// TwinCAT 3 PLC project Lampara_PLC
// ProgramVersion: 3.1.4024.0
// libraries:
//   Tc2_Standard, * (Beckhoff Automation GmbH)
//   Tc2_System, * (Beckhoff Automation GmbH)
//   Tc3_Module, * (Beckhoff Automation GmbH)
//   VisuDialogs, * (System)
// project tree:
//   / GlobalTextList.TcGTLO, PlcTask.TcTTO, Visualization Manager.TcVMO (not stored)
//   POUs/IL/ FB_LamparaAsignada_IL.TcPOU, FB_LamparaComputada_IL.TcPOU, FB_LamparaConmutada_IL.TcPOU, FB_LamparaIntermitente_IL.TcPOU, FB_LamparaMemorizada_IL.TcPOU, FB_LamparaTemporizada_IL.TcPOU, FB_LamparaTemporizada_IL_2.TcPOU
//   POUs/LD/ FB_LamparaAsignada_LD.TcPOU, FB_LamparaComputada_LD.TcPOU, FB_LamparaConmutada_LD.TcPOU, FB_LamparaConmutada_LD_2.TcPOU, FB_LamparaIntermitente_LD.TcPOU, FB_LamparaMemorizada_LD.TcPOU, FB_LamparaMemorizada_LD_2.TcPOU, FB_LamparaTemporizada_LD.TcPOU, FB_LamparaTemporizada_LD_2.TcPOU
//   POUs/ MAIN.TcPOU
//   POUs/SFC/ FB_LamparaAsignada_SFC.TcPOU, FB_LamparaAsignada_SFC_2.TcPOU, FB_LamparaComputada_SFC.TcPOU, FB_LamparaConmutada_SFC.TcPOU, FB_LamparaConmutada_SFC_2.TcPOU, FB_LamparaIntermitente_SFC.TcPOU, FB_LamparaIntermitente_SFC_2.TcPOU, FB_LamparaMemorizada_SFC.TcPOU, FB_LamparaMemorizada_SFC_2.TcPOU, FB_LamparaTemporizada_SFC.TcPOU, FB_LamparaTemporizada_SFC_2.TcPOU
//   POUs/ST/ FB_LamparaAsignada_ST.TcPOU, FB_LamparaComputada_ST.TcPOU, FB_LamparaConmutada_ST.TcPOU, FB_LamparaIntermitente_ST.TcPOU, FB_LamparaMemorizada_ST.TcPOU, FB_LamparaTemporizada_ST.TcPOU, FB_LamparaTemporizada_ST_2.TcPOU, FB_LamparaTemporizada_ST_3.TcPOU
//   VISUs/ VISU_Lampara.TcVIS
// real-time tasks:
//   TASK PlcTask: cycle T#10ms, priority 20, ADS port 350
//   TASK PlcTask1: cycle T#10ms, priority 21, ADS port 351

CONFIGURATION Lampara_PLC
    RESOURCE PLC ON TwinCAT3
        TASK PlcTask(INTERVAL := T#10ms, PRIORITY := 20);
        PROGRAM MAIN WITH PlcTask : MAIN;
    END_RESOURCE
END_CONFIGURATION

// ---- POUs/MAIN.TcPOU
PROGRAM MAIN
(*
 * =================================================================================
 * POU Nombre:      MAIN
 * File:            MAIN.TcPOU
 * Version:         1.0.0
 * Date:            2025-10-20
 * Author:          Victor Torres
 * ---------------------------------------------------------------------------------
 * Copyright (C) 2020-2025 Victor Torres
 * License:         GNU General Public License (GPL)
 * This program is free software; see the file "LICENSE" for details
 * ---------------------------------------------------------------------------------
 * Historial de Revisiones:
 * ------------------------
 * 1.0.0 - 2025-10-20 - VTL: Versión inicial
 * 0.1.0 - 2020-05-02 - VTL: Creacion
 * =================================================================================
 *)
 
 (*!
 * @brief MAIN: Programa Principal de TC3_Lampara
 *
 * @description
 * Ejemplo sencillo para mostras el uso de los elementos fundamentales de la libreria 
 * STANDARD del IEC 61131-3 en los diferentes lenguajes de la norma.
 *
 * 1. Lampara asignada     - la lampara "copia" el estado del pulsador
 * 2. Lampara memoriazada  - un pulsador enciende la lampara y otro la apaga
 * 3. Lampara conmutada    - el mismo pulsador enciende y apaga la lampara
 * 4. Lampara temporizada  - la lampara se apaga transcurrido un cierto tiempo
 *                           despues de accionar el pulsador
 * 5. Lampara intermitente - la lampara parpadea
 * 6. Lampara computada    - la lampara se enciende tras accionar varias veces el 
 *                           pulsador y se apaga al accionar el pulsador de reinicio
*)
 
VAR
    Lampara   AT %Q*  : BOOL;
    Pulsador  AT %I*  : BOOL;
    
// Definir lo que corresponda {LENGUAJE_IL, LENGUAJE_LD, LENGUAJE_ST, LENGUAJE_SFC}
{define LENGUAJE_SFC}
{IF defined(LENGUAJE_IL)}
    LamparaAsignada      : FB_LamparaAsignada_IL;
    LamparaMemorizada    : FB_LamparaMemorizada_IL;
    LamparaConmutada     : FB_LamparaConmutada_IL;
    LamparaTemporizada   : FB_LamparaTemporizada_IL;
    LamparaIntermitente  : FB_LamparaIntermitente_IL;
    LamparaComputada     : FB_LamparaComputada_IL;
{ELSIF defined(LENGUAJE_LD)}
    LamparaAsignada      : FB_LamparaAsignada_LD;
    LamparaMemorizada    : FB_LamparaMemorizada_LD;
    LamparaConmutada     : FB_LamparaConmutada_LD;
    LamparaTemporizada   : FB_LamparaTemporizada_LD;
    LamparaIntermitente  : FB_LamparaIntermitente_LD;
    LamparaComputada     : FB_LamparaComputada_LD;
{ELSIF defined(LENGUAJE_ST)}
    LamparaAsignada      : FB_LamparaAsignada_ST;
    LamparaMemorizada    : FB_LamparaMemorizada_ST;
    LamparaConmutada     : FB_LamparaConmutada_ST;
    LamparaTemporizada   : FB_LamparaTemporizada_ST_3;
    LamparaIntermitente  : FB_LamparaIntermitente_ST;
    LamparaComputada     : FB_LamparaComputada_ST;
{ELSIF defined(LENGUAJE_SFC)}
    LamparaAsignada      : FB_LamparaAsignada_SFC;
    LamparaMemorizada    : FB_LamparaMemorizada_SFC;
    LamparaConmutada     : FB_LamparaConmutada_SFC;
    LamparaTemporizada   : FB_LamparaTemporizada_SFC;
    LamparaIntermitente  : FB_LamparaIntermitente_SFC_2;
    LamparaComputada     : FB_LamparaComputada_SFC;
{END_IF}
END_VAR

Lampara := Pulsador;

LamparaAsignada();
LamparaMemorizada();
LamparaConmutada();
LamparaTemporizada();
LamparaComputada();
LamparaIntermitente();

END_PROGRAM

// ---- POUs/IL/FB_LamparaAsignada_IL.TcPOU
FUNCTION_BLOCK FB_LamparaAsignada_IL
// La lampara se enciende mientras se acciona el pulsador
VAR
    Lampara   AT %Q*  : BOOL;
    Pulsador  AT %I*  : BOOL;
END_VAR

// NETWORK 1
// instruction list
LD      Pulsador
ST      Lampara

END_FUNCTION_BLOCK

// ---- POUs/IL/FB_LamparaMemorizada_IL.TcPOU
FUNCTION_BLOCK FB_LamparaMemorizada_IL
// La lampara se enciende al accionar el pulsador de conexion
// La lampara se apaga al accionar el pulsador de desconexion
VAR
    Lampara              AT %Q*  : BOOL;
    PulsadorConexion     AT %I*  : BOOL;
    PulsadorDesconexion  AT %I*  : BOOL;
END_VAR

// NETWORK 1
// instruction list
LD      PulsadorConexion
S       Lampara
LD      PulsadorDesconexion
R       Lampara

END_FUNCTION_BLOCK

// ---- POUs/IL/FB_LamparaConmutada_IL.TcPOU
FUNCTION_BLOCK FB_LamparaConmutada_IL
// La lampara se enciende si estando apagada se acciona el pulsador
// La lampara se apaga si estando encendida se acciona el pulsador
VAR
    Pulsacion         : R_TRIG;
    Lampara   AT %Q*  : BOOL;
    Pulsador  AT %I*  : BOOL;
END_VAR

// NETWORK 1
// instruction list
CAL     Pulsacion(
    CLK     := Pulsador)

// NETWORK 2
// instruction list
LD      Pulsacion.Q
JMPCN   End

// NETWORK 3
// instruction list
LDN     Lampara
ST      Lampara

// NETWORK 4
End:
// instruction list

END_FUNCTION_BLOCK

// ---- POUs/IL/FB_LamparaTemporizada_IL.TcPOU
FUNCTION_BLOCK FB_LamparaTemporizada_IL
// La lampara se enciende al accionar el pulsador
// La lampara se apaga transcurrido un tiempo encendidaVAR_INPUT
VAR
    TiempoEncendido   : TIME := T#2S;
END_VAR
VAR_OUTPUT
    TiempoPendiente   : TIME;
END_VAR
VAR
    Temporizador      : TON;
    Lampara   AT %Q*  : BOOL;
    Pulsador  AT %I*  : BOOL;
END_VAR

// NETWORK 1
// instruction list
CAL     Temporizador(
    IN      := Lampara,
    PT      := TiempoEncendido)

// NETWORK 2
// instruction list
LD      TiempoEncendido
SUB     Temporizador.ET
ST      TiempoPendiente

// NETWORK 3
// instruction list
LD      Pulsador
S       Lampara

// NETWORK 4
// instruction list
LD      Temporizador.Q
R       Lampara

END_FUNCTION_BLOCK

// ---- POUs/IL/FB_LamparaIntermitente_IL.TcPOU
FUNCTION_BLOCK FB_LamparaIntermitente_IL
// La lampara parpadea de forma continua
VAR_INPUT
    TiempoParpadeo   : TIME := T#500MS;
END_VAR
VAR
    Temporizador     : TON;
    Lampara  AT %Q*  : BOOL;
END_VAR

// NETWORK 1
// Temporizador auto-pilotado
// instruction list
CAL     Temporizador(
    IN      := NOT Temporizador.Q
    PT      := TiempoParpadeo)

// NETWORK 2
// instruction list
LD      Temporizador.Q
JMPCN   End

// NETWORK 3
// Salida conmutada
// instruction list
LD      Lampara
STN     Lampara

// NETWORK 4
End:
// instruction list

END_FUNCTION_BLOCK

// ---- POUs/IL/FB_LamparaComputada_IL.TcPOU
FUNCTION_BLOCK FB_LamparaComputada_IL
// La lampara se enciende tras un determinado numero de pulsaciones
// La lampara se apaga tras accionar el pulsador de reinicio
VAR_INPUT
    ManiobrasTotales     : UINT := 2;
END_VAR
VAR_OUTPUT
    ManiobrasPendientes  : UINT;
END_VAR
VAR
    Contador                  : CTD := (CV := ManiobrasTotales);
    Lampara           AT %Q*  : BOOL;
    Pulsador          AT %I*  : BOOL;
    PulsadorReinicio  AT %I*  : BOOL;
END_VAR

// NETWORK 1
// instruction list
CAL     Contador(
    CD      := Pulsador,
    LOAD    := PulsadorReinicio,
    PV      := ManiobrasTotales)

// NETWORK 2
// instruction list
LD      Contador.Q
ST      Lampara

// NETWORK 3
// instruction list
LD      Contador.CV
ST      ManiobrasPendientes

END_FUNCTION_BLOCK

// ---- POUs/LD/FB_LamparaAsignada_LD.TcPOU
FUNCTION_BLOCK FB_LamparaAsignada_LD
// La lampara se enciende mientras se acciona el pulsador
VAR
    Lampara   AT %Q*  : BOOL;
    Pulsador  AT %I*  : BOOL;
END_VAR

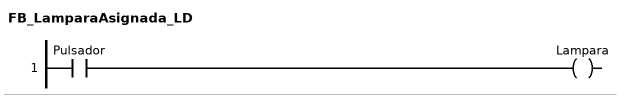
// NETWORK 1
Lampara := Pulsador;

END_FUNCTION_BLOCK

// ---- POUs/LD/FB_LamparaMemorizada_LD.TcPOU
FUNCTION_BLOCK FB_LamparaMemorizada_LD
// La lampara se enciende al accionar el pulsador de conexion
// La lampara se apaga al accionar el pulsador de desconexion
VAR
    Lampara              AT %Q*  : BOOL;
    PulsadorConexion     AT %I*  : BOOL;
    PulsadorDesconexion  AT %I*  : BOOL;
END_VAR

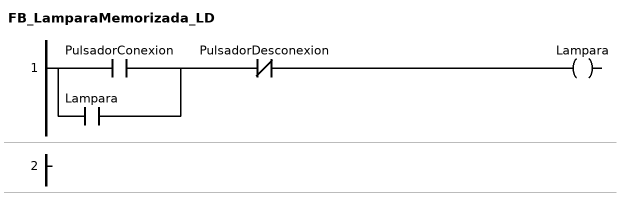
// NETWORK 1
Lampara := (PulsadorConexion OR Lampara) AND NOT PulsadorDesconexion;

// NETWORK 2

END_FUNCTION_BLOCK

// ---- POUs/LD/FB_LamparaConmutada_LD.TcPOU
FUNCTION_BLOCK FB_LamparaConmutada_LD
// La lampara se enciende si estando apagada se acciona el pulsador
// La lampara se apaga si estando encendida se acciona el pulsador
VAR
    Pulsacion         : R_TRIG;
    Lampara   AT %Q*  : BOOL;
    Pulsador  AT %I*  : BOOL;
END_VAR

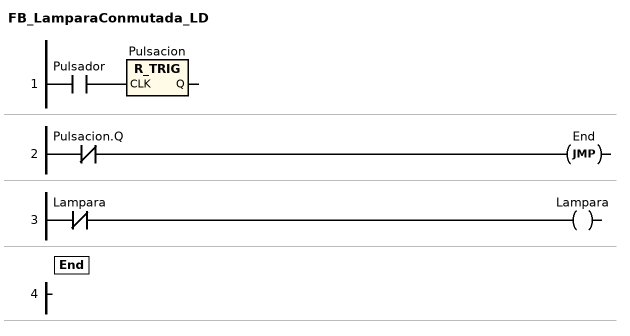
// NETWORK 1
Pulsacion(CLK := Pulsador); // R_TRIG

// NETWORK 2
IF NOT Pulsacion.Q THEN JMP End; END_IF

// NETWORK 3
Lampara := NOT Lampara;

// NETWORK 4
End: ;

END_FUNCTION_BLOCK

// ---- POUs/LD/FB_LamparaTemporizada_LD.TcPOU
FUNCTION_BLOCK FB_LamparaTemporizada_LD
// La lampara se enciende al accionar el pulsador
// La lampara se apaga transcurrido un tiempo encendida
VAR_INPUT
    TiempoEncendido   : TIME := T#2S;
END_VAR
VAR_OUTPUT
    TiempoPendiente   : TIME;
END_VAR
VAR
    Temporizador      : TON;
    Memoria           : RS;
    Lampara   AT %Q*  : BOOL;
    Pulsador  AT %I*  : BOOL;
END_VAR

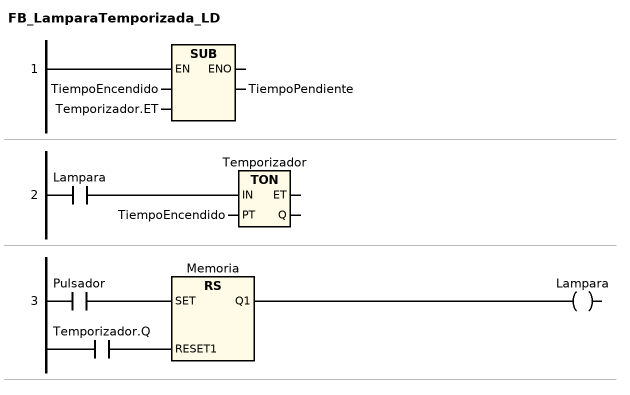
// NETWORK 1
TiempoPendiente := TiempoEncendido - Temporizador.ET;

// NETWORK 2
Temporizador(IN := Lampara, PT := TiempoEncendido); // TON

// NETWORK 3
Memoria(SET := Pulsador, RESET1 := Temporizador.Q); // RS
Lampara := Memoria.Q1;

END_FUNCTION_BLOCK

// ---- POUs/LD/FB_LamparaIntermitente_LD.TcPOU
FUNCTION_BLOCK FB_LamparaIntermitente_LD
// La lampara parpadea de forma continua
VAR_INPUT
    TiempoParpadeo   : TIME := T#500MS;
END_VAR
VAR
    Temporizador     : TON;
    Lampara  AT %Q*  : BOOL;
END_VAR

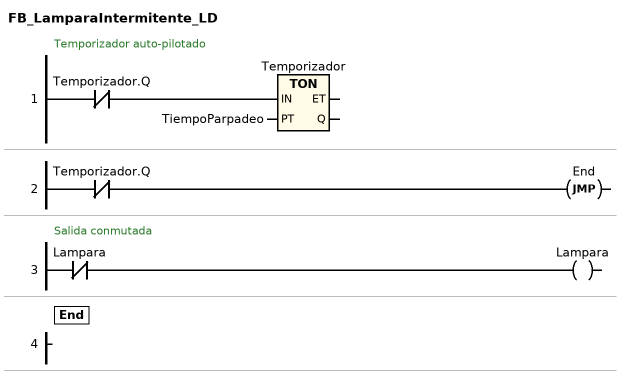
// NETWORK 1
// Temporizador auto-pilotado
Temporizador(IN := NOT Temporizador.Q, PT := TiempoParpadeo); // TON

// NETWORK 2
IF NOT Temporizador.Q THEN JMP End; END_IF

// NETWORK 3
// Salida conmutada
Lampara := NOT Lampara;

// NETWORK 4
End: ;

END_FUNCTION_BLOCK

// ---- POUs/LD/FB_LamparaComputada_LD.TcPOU
FUNCTION_BLOCK FB_LamparaComputada_LD
// La lampara se enciende tras un determinado numero de pulsaciones
// La lampara se apaga tras accionar el pulsador de reinicio
VAR_INPUT
    ManiobrasTotales     : UINT := 2;
END_VAR
VAR_OUTPUT
    ManiobrasPendientes  : UINT;
END_VAR
VAR
    Contador                  : CTD := (CV := ManiobrasTotales);
    Lampara           AT %Q*  : BOOL;
    Pulsador          AT %I*  : BOOL;
    PulsadorReinicio  AT %I*  : BOOL;
END_VAR

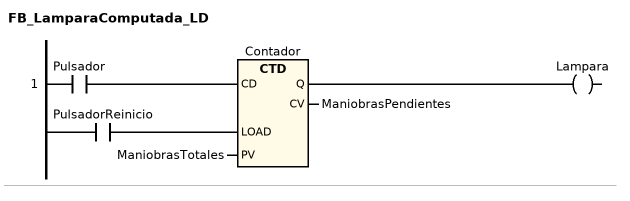
// NETWORK 1
Contador(CD := Pulsador, LOAD := PulsadorReinicio, PV := ManiobrasTotales, CV => ManiobrasPendientes); // CTD
Lampara := Contador.Q;

END_FUNCTION_BLOCK

// ---- POUs/ST/FB_LamparaAsignada_ST.TcPOU
FUNCTION_BLOCK FB_LamparaAsignada_ST
// La lampara se enciende mientras se acciona el pulsador
VAR
    Lampara  AT %Q* : BOOL;
    Pulsador AT %I* : BOOL;
END_VAR

Lampara := Pulsador;

END_FUNCTION_BLOCK

// ---- POUs/ST/FB_LamparaMemorizada_ST.TcPOU
FUNCTION_BLOCK FB_LamparaMemorizada_ST
// La lampara se enciende al accionar el pulsador de conexion
// La lampara se apaga al accionar el pulsador de desconexion
VAR
    Lampara              AT %Q*  : BOOL;
    PulsadorConexion     AT %I*  : BOOL;
    PulsadorDesconexion  AT %I*  : BOOL;
END_VAR

IF PulsadorDesconexion THEN
    Lampara := FALSE;
ELSIF PulsadorConexion THEN
    Lampara := TRUE;
END_IF;

END_FUNCTION_BLOCK

// ---- POUs/ST/FB_LamparaConmutada_ST.TcPOU
FUNCTION_BLOCK FB_LamparaConmutada_ST
// La lampara se enciende si estando apagada se acciona el pulsador
// La lampara se apaga si estando encendida se acciona el pulsador
VAR
    Pulsacion         : R_TRIG;
    Lampara   AT %Q*  : BOOL;
    Pulsador  AT %I*  : BOOL;
END_VAR

Pulsacion(CLK := Pulsador);

IF Pulsacion.Q THEN
    Lampara := NOT Lampara;
END_IF;

END_FUNCTION_BLOCK

// ---- POUs/ST/FB_LamparaTemporizada_ST_3.TcPOU
FUNCTION_BLOCK FB_LamparaTemporizada_ST_3
// Lampara temporizada con tiempo prolongado con incremento variable
VAR_INPUT
    TiempoEncendido   : TIME := T#2S;
    IncrementoTiempo  : TIME := T#1S;
END_VAR
VAR_OUTPUT
    TiempoPendiente   : TIME;
END_VAR
VAR
    Temporizador      : TON;
    FlancoPulsador    : R_TRIG;
    TiempoActual      : TIME;

    Lampara   AT %Q*  : BOOL;
    Pulsador  AT %I*  : BOOL;
END_VAR

FlancoPulsador(CLK := Pulsador);

Temporizador(
    IN := Lampara AND NOT Pulsador, 
    PT := TiempoActual
    );

IF (Lampara AND FlancoPulsador.Q) THEN
    TiempoActual := TiempoActual + IncrementoTiempo;
ELSIF (NOT Lampara AND FlancoPulsador.Q) THEN
    TiempoActual := TiempoEncendido;
END_IF;

IF Pulsador THEN
    Lampara := TRUE;
ELSIF Temporizador.Q THEN
    Lampara := FALSE;
END_IF;

TiempoPendiente := TiempoActual - Temporizador.ET;

END_FUNCTION_BLOCK

// ---- POUs/ST/FB_LamparaIntermitente_ST.TcPOU
FUNCTION_BLOCK FB_LamparaIntermitente_ST
// La lampara parpadea de forma continua
VAR_INPUT
    TiempoParpadeo   : TIME := T#500MS;
END_VAR
VAR
    Temporizador     : TON;
    Lampara  AT %Q*  : BOOL;
END_VAR

// Temporizador auto-pilotado
Temporizador(
    IN := NOT Temporizador.Q,
    PT := TiempoParpadeo
    );

// Salida conmutada
IF Temporizador.Q THEN
    Lampara := NOT Lampara;
END_IF;

END_FUNCTION_BLOCK

// ---- POUs/ST/FB_LamparaComputada_ST.TcPOU
FUNCTION_BLOCK FB_LamparaComputada_ST
// La lampara se enciende tras un determinado numero de pulsaciones
// La lampara se apaga tras accionar el pulsador de reinicio
VAR_INPUT
    ManiobrasTotales     : UINT := 2;
END_VAR
VAR_OUTPUT
    ManiobrasPendientes  : UINT;
END_VAR
VAR
    Contador  : CTD := (CV := ManiobrasTotales);
    
    Lampara           AT %Q*  : BOOL;
    Pulsador          AT %I*  : BOOL;
    PulsadorReinicio  AT %I*  : BOOL;
END_VAR

Contador(
    CD   := Pulsador,
    LOAD := PulsadorReinicio,
    PV   := ManiobrasTotales,
    Q    => Lampara,
    CV   => ManiobrasPendientes
    );

END_FUNCTION_BLOCK

// ---- POUs/SFC/FB_LamparaAsignada_SFC.TcPOU
FUNCTION_BLOCK FB_LamparaAsignada_SFC
// La lampara se enciende mientras se acciona el pulsador
VAR
    Lampara   AT %Q*  : BOOL;
    Pulsador  AT %I*  : BOOL;
END_VAR

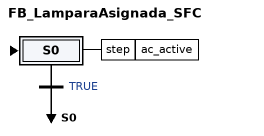
INITIAL_STEP S0:
    ac_active(N);  // step action
END_STEP
TRANSITION FROM S0 TO S0
    := TRUE;
END_TRANSITION

ACTION ac_active:
Lampara := S0.x AND Pulsador;
END_ACTION

END_FUNCTION_BLOCK

// ---- POUs/SFC/FB_LamparaMemorizada_SFC.TcPOU
FUNCTION_BLOCK FB_LamparaMemorizada_SFC
// La lampara se enciende al accionar el pulsador de conexion
// La lampara se apaga al accionar el pulsador de desconexion
VAR
    Lampara              AT %Q*  : BOOL;
    PulsadorConexion     AT %I*  : BOOL;
    PulsadorDesconexion  AT %I*  : BOOL;
END_VAR

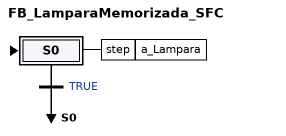
INITIAL_STEP S0:
    a_Lampara(N);  // step action
END_STEP
TRANSITION FROM S0 TO S0
    := TRUE;
END_TRANSITION

ACTION a_Lampara:
IF PulsadorDesconexion THEN
    Lampara := FALSE;
ELSIF PulsadorConexion THEN
    Lampara := TRUE;
END_IF;
END_ACTION

END_FUNCTION_BLOCK

// ---- POUs/SFC/FB_LamparaConmutada_SFC.TcPOU
FUNCTION_BLOCK FB_LamparaConmutada_SFC
// La lampara se enciende tras un determinado numero de pulsaciones
// La lampara se apaga tras accionar el pulsador de reinicio
VAR
    Pulsacion         : R_TRIG;
    Lampara   AT %Q*  : BOOL;
    Pulsador  AT %I*  : BOOL;
END_VAR

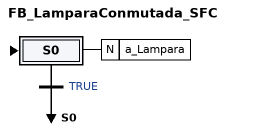
INITIAL_STEP S0:
    a_Lampara(N);
END_STEP
TRANSITION FROM S0 TO S0
    := TRUE;
END_TRANSITION

ACTION a_Lampara:
Pulsacion(CLK := Pulsador);

IF Pulsacion.Q THEN
    Lampara := NOT Lampara;
END_IF;
END_ACTION

END_FUNCTION_BLOCK

// ---- POUs/SFC/FB_LamparaTemporizada_SFC.TcPOU
FUNCTION_BLOCK FB_LamparaTemporizada_SFC
// La lampara se enciende al accionar el pulsador
// La lampara se apaga transcurrido un tiempo encendida
VAR_INPUT
    TiempoEncendido   : TIME := T#2S;
END_VAR
VAR_OUTPUT
    TiempoPendiente   : TIME;
END_VAR
VAR
    Lampara   AT %Q*  : BOOL;
    Pulsador  AT %I*  : BOOL;
END_VAR

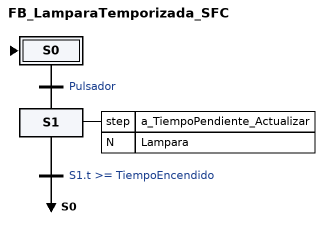
INITIAL_STEP S0:
END_STEP
TRANSITION FROM S0 TO S1
    := Pulsador;
END_TRANSITION
STEP S1:
    a_TiempoPendiente_Actualizar(N);  // step action
    Lampara(N);
END_STEP
TRANSITION FROM S1 TO S0
    := S1.t >= TiempoEncendido;
END_TRANSITION

ACTION a_TiempoPendiente_Actualizar:
TiempoPendiente := TiempoEncendido - S1.t;
END_ACTION

END_FUNCTION_BLOCK

// ---- POUs/SFC/FB_LamparaIntermitente_SFC_2.TcPOU
FUNCTION_BLOCK FB_LamparaIntermitente_SFC_2
// La lampara parpadea de forma continua
VAR_INPUT
    TiempoParpadeo   : TIME := T#500MS;
END_VAR
VAR
    Lampara  AT %Q*  : BOOL;
END_VAR

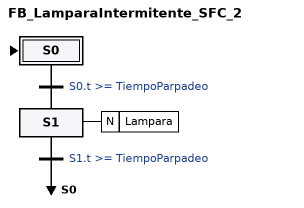
INITIAL_STEP S0:
END_STEP
TRANSITION FROM S0 TO S1
    := S0.t >= TiempoParpadeo;
END_TRANSITION
STEP S1:
    Lampara(N);
END_STEP
TRANSITION FROM S1 TO S0
    := S1.t >= TiempoParpadeo;
END_TRANSITION

END_FUNCTION_BLOCK

// ---- POUs/SFC/FB_LamparaComputada_SFC.TcPOU
FUNCTION_BLOCK FB_LamparaComputada_SFC
// La lampara se enciende tras un determinado numero de pulsaciones
// La lampara se apaga tras accionar el pulsador de reinicio
VAR_INPUT
    ManiobrasTotales        : UINT := 2;
END_VAR
VAR_OUTPUT
    ManiobrasPendientes     : UINT := ManiobrasTotales;
END_VAR
VAR
    FlancoPulsador          : R_TRIG;
    Lampara           AT %Q*: BOOL;
    Pulsador          AT %I*: BOOL;
    PulsadorReinicio  AT %I*  : BOOL;
END_VAR

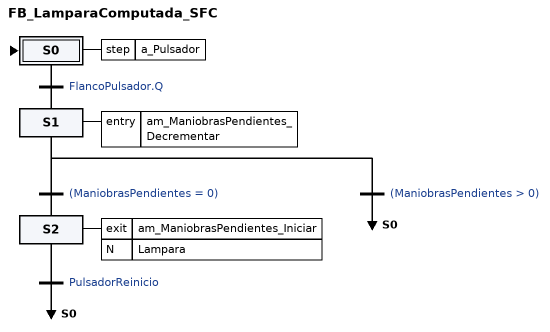
INITIAL_STEP S0:
    a_Pulsador(N);  // step action
END_STEP
TRANSITION FROM S0 TO S1
    := FlancoPulsador.Q;
END_TRANSITION
STEP S1:
    am_ManiobrasPendientes_Decrementar(P1);  // entry action
END_STEP
TRANSITION FROM S1 TO S2
    := (ManiobrasPendientes = 0);
END_TRANSITION
TRANSITION FROM S1 TO S0
    := (ManiobrasPendientes > 0);
END_TRANSITION
STEP S2:
    am_ManiobrasPendientes_Iniciar(P0);  // exit action
    Lampara(N);
END_STEP
TRANSITION FROM S2 TO S0
    := PulsadorReinicio;
END_TRANSITION

ACTION a_Pulsador:
FlancoPulsador(CLK := Pulsador);
END_ACTION

ACTION am_ManiobrasPendientes_Decrementar:
IF (ManiobrasPendientes > 0) THEN 
    ManiobrasPendientes := ManiobrasPendientes - 1;
END_IF;
END_ACTION

ACTION am_ManiobrasPendientes_Iniciar:
ManiobrasPendientes := ManiobrasTotales;
END_ACTION

END_FUNCTION_BLOCK

// ---- POUs/IL/FB_LamparaTemporizada_IL_2.TcPOU
FUNCTION_BLOCK FB_LamparaTemporizada_IL_2
// Lampara temporizada con tiempo de espera prolongado
VAR_INPUT
    TiempoEncendido   : TIME := T#2S;
END_VAR
VAR_OUTPUT
    TiempoPendiente   : TIME;
END_VAR
VAR
    Temporizador      : TON;
    Lampara   AT %Q*  : BOOL;
    Pulsador  AT %I*  : BOOL;
END_VAR

// NETWORK 1
// instruction list
CAL     Temporizador(
    IN      := NOT Pulsador AND Lampara,
    PT      := TiempoEncendido)

// NETWORK 2
// instruction list
LD      TiempoEncendido
SUB     Temporizador.ET
ST      TiempoPendiente

// NETWORK 3
// instruction list
LD      Pulsador
S       Lampara

// NETWORK 4
// instruction list
LD      Temporizador.Q
R       Lampara

// NETWORK 5

END_FUNCTION_BLOCK

// ---- POUs/LD/FB_LamparaConmutada_LD_2.TcPOU
FUNCTION_BLOCK FB_LamparaConmutada_LD_2
// La lampara se enciende si estando apagada se acciona el pulsador
// La lampara se apaga si estando encendida se acciona el pulsador
VAR
    Pulsacion         : R_TRIG;
    MemoriaLampara    : BOOL;
    Lampara   AT %Q*  : BOOL;
    Pulsador  AT %I*  : BOOL;
END_VAR

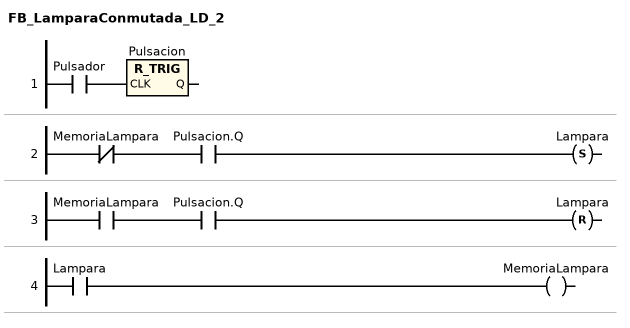
// NETWORK 1
Pulsacion(CLK := Pulsador); // R_TRIG

// NETWORK 2
Lampara S= NOT MemoriaLampara AND Pulsacion.Q;

// NETWORK 3
Lampara R= MemoriaLampara AND Pulsacion.Q;

// NETWORK 4
MemoriaLampara := Lampara;

END_FUNCTION_BLOCK

// ---- POUs/LD/FB_LamparaMemorizada_LD_2.TcPOU
FUNCTION_BLOCK FB_LamparaMemorizada_LD_2
// La lampara se enciende al accionar el pulsador de conexion
// La lampara se apaga al accionar el pulsador de desconexion
VAR
    Memoria                      : RS;
    Lampara              AT %Q*  : BOOL;
    PulsadorConexion     AT %I*  : BOOL;
    PulsadorDesconexion  AT %I*  : BOOL;
END_VAR

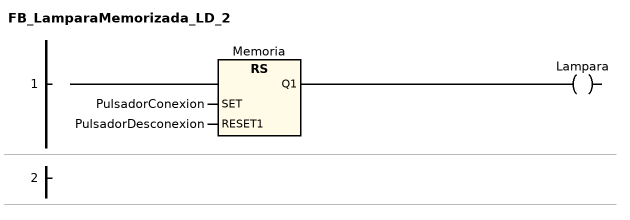
// NETWORK 1
Memoria(SET := PulsadorConexion, RESET1 := PulsadorDesconexion); // RS
Lampara := Memoria.Q1;

// NETWORK 2

END_FUNCTION_BLOCK

// ---- POUs/LD/FB_LamparaTemporizada_LD_2.TcPOU
FUNCTION_BLOCK FB_LamparaTemporizada_LD_2
// Lampara temporizada con tiempo de espera prolongado
VAR_INPUT
    TiempoEncendido   : TIME := T#2S;
    IncrementoTiempo  : TIME := T#1S;
END_VAR
VAR_OUTPUT
    TiempoPendiente   : TIME;
END_VAR
VAR
    Temporizador      : TON;
    Memoria           : RS;
    Lampara   AT %Q*  : BOOL;
    Pulsador  AT %I*  : BOOL;
END_VAR

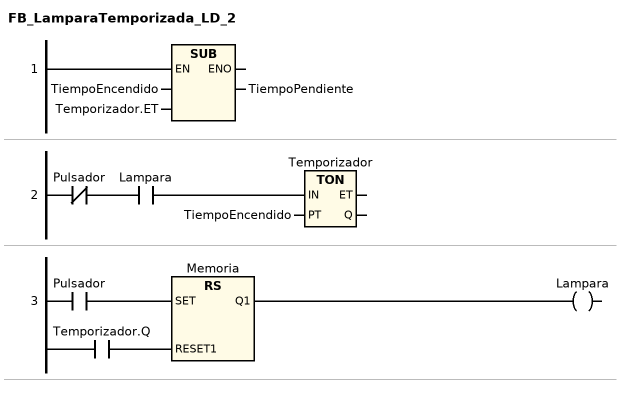
// NETWORK 1
TiempoPendiente := TiempoEncendido - Temporizador.ET;

// NETWORK 2
Temporizador(IN := NOT Pulsador AND Lampara, PT := TiempoEncendido); // TON

// NETWORK 3
Memoria(SET := Pulsador, RESET1 := Temporizador.Q); // RS
Lampara := Memoria.Q1;

END_FUNCTION_BLOCK

// ---- POUs/SFC/FB_LamparaAsignada_SFC_2.TcPOU
FUNCTION_BLOCK FB_LamparaAsignada_SFC_2
// La lampara se enciende mientras se acciona el pulsador
VAR
    Lampara   AT %Q*  : BOOL;
    Pulsador  AT %I*  : BOOL;
END_VAR

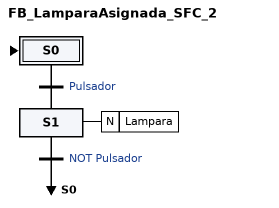
INITIAL_STEP S0:
END_STEP
TRANSITION FROM S0 TO S1
    := Pulsador;
END_TRANSITION
STEP S1:
    Lampara(N);
END_STEP
TRANSITION FROM S1 TO S0
    := NOT Pulsador;
END_TRANSITION

END_FUNCTION_BLOCK

// ---- POUs/SFC/FB_LamparaConmutada_SFC_2.TcPOU
FUNCTION_BLOCK FB_LamparaConmutada_SFC_2
// La lampara se enciende si estando apagada se acciona el pulsador
// La lampara se apaga si estando encendida se acciona el pulsador
VAR
    Pulsacion         : R_TRIG;
    Lampara   AT %Q*  : BOOL;
    Pulsador  AT %I*  : BOOL;
END_VAR

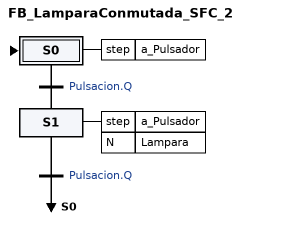
INITIAL_STEP S0:
    a_Pulsador(N);  // step action
END_STEP
TRANSITION FROM S0 TO S1
    := Pulsacion.Q;
END_TRANSITION
STEP S1:
    a_Pulsador(N);  // step action
    Lampara(N);
END_STEP
TRANSITION FROM S1 TO S0
    := Pulsacion.Q;
END_TRANSITION

ACTION a_Pulsador:
Pulsacion(CLK := Pulsador);
END_ACTION

END_FUNCTION_BLOCK

// ---- POUs/SFC/FB_LamparaIntermitente_SFC.TcPOU
FUNCTION_BLOCK FB_LamparaIntermitente_SFC
// La lampara parpadea de forma continua
VAR_INPUT
    TiempoParpadeo  : TIME := T#500MS;
END_VAR
VAR
    TiempoAnterior  : TIME;
    
    Lampara AT %Q*  : BOOL;
END_VAR

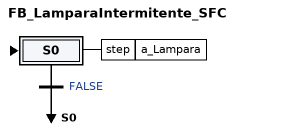
INITIAL_STEP S0:
    a_Lampara(N);  // step action
END_STEP
TRANSITION FROM S0 TO S0
    := FALSE;
END_TRANSITION

ACTION a_Lampara:
IF S0.t - TiempoAnterior > TiempoParpadeo THEN
    Lampara := NOT Lampara;
    TiempoAnterior := S0.t;
END_IF;
END_ACTION

END_FUNCTION_BLOCK

// ---- POUs/SFC/FB_LamparaMemorizada_SFC_2.TcPOU
FUNCTION_BLOCK FB_LamparaMemorizada_SFC_2
// La lampara se enciende al accionar el pulsador de conexion
// La lampara se apaga al accionar el pulsador de desconexion
VAR
    Lampara              AT %Q*  : BOOL;
    PulsadorConexion     AT %I*  : BOOL;
    PulsadorDesconexion  AT %I*  : BOOL;
END_VAR

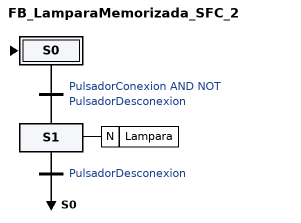
INITIAL_STEP S0:
END_STEP
TRANSITION FROM S0 TO S1
    := PulsadorConexion AND NOT PulsadorDesconexion;
END_TRANSITION
STEP S1:
    Lampara(N);
END_STEP
TRANSITION FROM S1 TO S0
    := PulsadorDesconexion;
END_TRANSITION

END_FUNCTION_BLOCK

// ---- POUs/SFC/FB_LamparaTemporizada_SFC_2.TcPOU
FUNCTION_BLOCK FB_LamparaTemporizada_SFC_2
// Lampara temporizada con tiempo de espera prolongado
VAR_INPUT
    TiempoEncendido   : TIME := T#2S;
    IncrementoTiempo  : TIME := T#1S;
END_VAR
VAR_OUTPUT
    TiempoPendiente   : TIME;
END_VAR
VAR
    Lampara   AT %Q*  : BOOL;
    Pulsador  AT %I*  : BOOL;
END_VAR

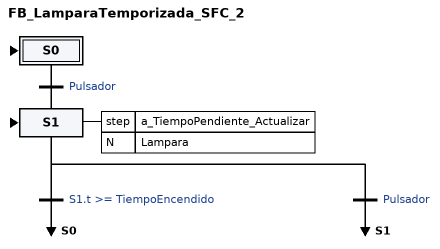
INITIAL_STEP S0:
END_STEP
TRANSITION FROM S0 TO S1
    := Pulsador;
END_TRANSITION
STEP S1:
    a_TiempoPendiente_Actualizar(N);  // step action
    Lampara(N);
END_STEP
TRANSITION FROM S1 TO S0
    := S1.t >= TiempoEncendido;
END_TRANSITION
TRANSITION FROM S1 TO S1
    := Pulsador;
END_TRANSITION

ACTION a_TiempoPendiente_Actualizar:
TiempoPendiente := TiempoEncendido - S1.t;
END_ACTION

END_FUNCTION_BLOCK

// ---- POUs/ST/FB_LamparaTemporizada_ST.TcPOU
FUNCTION_BLOCK FB_LamparaTemporizada_ST
// La lampara se enciende al accionar el pulsador
// La lampara se apaga transcurrido un tiempo encendida
VAR_INPUT
    TiempoEncendido   : TIME := T#2S;
END_VAR
VAR_OUTPUT
    TiempoPendiente   : TIME;
END_VAR
VAR
    Temporizador      : TON;
    
    Lampara   AT %Q*  : BOOL;
    Pulsador  AT %I*  : BOOL;
END_VAR

Temporizador(
    IN := Lampara, 
    PT := TiempoEncendido
    );

IF Pulsador THEN
    Lampara := TRUE;
ELSIF Temporizador.Q THEN
    Lampara := FALSE;
END_IF;

TiempoPendiente := TiempoEncendido - Temporizador.ET;

END_FUNCTION_BLOCK

// ---- POUs/ST/FB_LamparaTemporizada_ST_2.TcPOU
FUNCTION_BLOCK FB_LamparaTemporizada_ST_2
// Lampara temporizada con tiempo de espera prolongado
VAR_INPUT
    TiempoEncendido   : TIME := T#2S;
VAR
VAR_OUTPUT
    TiempoPendiente   : TIME;
END_VAR
VAR
    Temporizador      : TON;
    
    Lampara   AT %Q*  : BOOL;
    Pulsador  AT %I*  : BOOL;
END_VAR

Temporizador(
    IN := Lampara AND NOT Pulsador,
    PT := TiempoEncendido
    );

IF Pulsador THEN
    Lampara := TRUE;
ELSIF Temporizador.Q THEN
    Lampara := FALSE;
END_IF;

TiempoPendiente := TiempoEncendido - Temporizador.ET;

END_FUNCTION_BLOCK

// ---- GlobalTextList.TcGTLO
TEXTLIST GlobalTextList
  279 = '%.2f [s]'
  147 = '%d'
  629 = '%t[ss:ms]'
  152 = '%t[ss]'
  948 = 'Apaga'
  32 = 'Asignada'
  589 = 'Computada'
  203 = 'Conmutada'
  701 = 'Enciende'
  703 = 'Habilitada'
  728 = 'Incremento'
  251 = 'Intermitente'
  961 = 'Lámpara'
  797 = 'MAIN'
  817 = 'Maniobras'
  591 = 'Memorizada'
  237 = 'Pendiente'
  884 = 'Pulsador'
  517 = 'Reinicia'
  167 = 'Temporizada'
  524 = 'Tiempo'
  250 = 'Total'
END_TEXTLIST

// ---- VISUs/VISU_Lampara.TcVIS
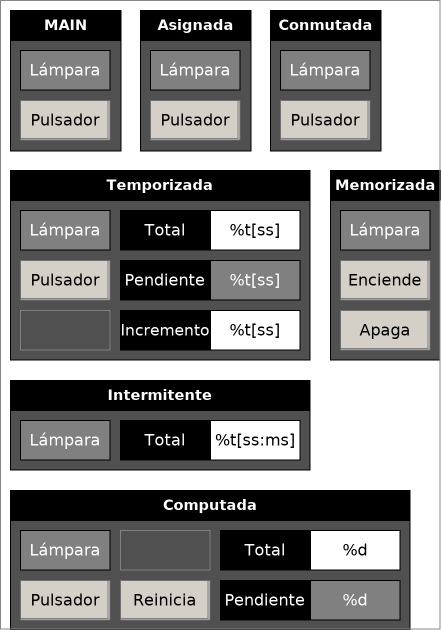
VISUALIZATION VISU_Lampara  // 441x630
    Rectangle (10,40 111x111)
    Rectangle (20,50 90x40), "Lámpara", colour toggle: MAIN.Lampara
    Button (20,100 90x40), "Pulsador"
        tap MAIN.Pulsador
    Rectangle (10,10 111x30), "MAIN"
    Rectangle (10,200 300x160)
    Rectangle (20,210 90x40), "Lámpara", colour toggle: MAIN.LamparaTemporizada.Lampara
    Button (20,260 90x40), "Pulsador"
        tap MAIN.LamparaTemporizada.Pulsador
    Rectangle (10,170 300x30), "Temporizada"
    Rectangle (120,210 90x40), "Total"
    Rectangle (210,210 90x40), "%t[ss]", text variable: MAIN.LamparaTemporizada.TiempoEncendido
        OnMouseDown: write the text variable via Default
    Rectangle (120,260 90x40), "Pendiente"
    Rectangle (210,260 90x40), "%t[ss]", text variable: MAIN.LamparaTemporizada.TiempoPendiente
    Rectangle (140,40 111x111)
    Rectangle (150,50 90x40), "Lámpara", colour toggle: MAIN.LamparaAsignada.Lampara
    Button (150,100 90x40), "Pulsador"
        tap MAIN.LamparaAsignada.Pulsador
    Rectangle (140,10 111x30), "Asignada"
    Rectangle (270,40 111x111)
    Rectangle (280,50 90x40), "Lámpara", colour toggle: MAIN.LamparaConmutada.Lampara
    Button (280,100 90x40), "Pulsador"
        tap MAIN.LamparaConmutada.Pulsador
    Rectangle (270,10 111x30), "Conmutada"
    Rectangle (10,520 400x110)
    Rectangle (20,530 90x40), "Lámpara", colour toggle: MAIN.LamparaComputada.Lampara
    Button (20,580 90x40), "Pulsador"
        tap MAIN.LamparaComputada.Pulsador
    Rectangle (10,490 400x30), "Computada"
    Rectangle (220,530 90x40), "Total"
    Rectangle (310,530 90x40), "%d", text variable: MAIN.LamparaComputada.ManiobrasTotales
        OnMouseDown: write the text variable via Default
    Rectangle (220,580 90x40), "Pendiente"
    Rectangle (310,580 90x40), "%d", text variable: MAIN.LamparaComputada.ManiobrasPendientes
    Button (120,580 90x40), "Reinicia"
        tap MAIN.LamparaComputada.PulsadorReinicio
    Rectangle (330,200 110x160)
    Rectangle (340,210 90x40), "Lámpara", colour toggle: MAIN.LamparaMemorizada.Lampara
    Button (340,310 90x40), "Apaga"
        tap MAIN.LamparaMemorizada.PulsadorDesconexion
    Rectangle (330,170 111x30), "Memorizada"
    Button (340,260 90x40), "Enciende"
        tap MAIN.LamparaMemorizada.PulsadorConexion
    Rectangle (10,410 300x60)
    Rectangle (20,420 90x40), "Lámpara", colour toggle: MAIN.LamparaIntermitente.Lampara
    Rectangle (10,380 300x30), "Intermitente"
    Rectangle (120,420 90x40), "Total"
    Rectangle (210,420 90x40), "%t[ss:ms]", text variable: MAIN.LamparaIntermitente.TiempoParpadeo
        OnMouseDown: write the text variable via Default
    Rectangle (120,310 90x40), "Incremento"
    Rectangle (210,310 90x40), "%t[ss]", text variable: MAIN.LamparaTemporizada.IncrementoTiempo
        OnMouseDown: write the text variable via Default
    Rectangle (120,530 90x40)
    Rectangle (20,310 90x40)
END_VISUALIZATION
